ABB RobotStudio station: SCM_ExampleStation.rspag

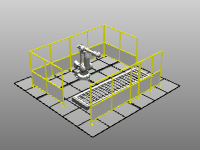
--- station ---
Station Station (saved by RobotStudio 6.4.7060.110)
Controller IRB4400_60_SCM_Example
  mechanical unit ROB_1: IRB4400_60_SCM_Example, 6 joints, base frame (0, 0, 0) mm
Layout (positions relative to the parent item):
  - Fence_2500 [graphiccomponentgroup, from Equipment\Fence_2500.rslib] at (-1042.5, 0, 0) mm
    - Body 1 [part, from Equipment\Fence_2500.rslib]
    - Body 2 [part, from Equipment\Fence_2500.rslib]
  - Fence_2500_2 [graphiccomponentgroup, from Equipment\Fence_2500.rslib] at (-1041.34, -2499.15, 0) mm
    - Body 1 [part, from Equipment\Fence_2500.rslib]
    - Body 2 [part, from Equipment\Fence_2500.rslib]
  - Fence_2500_3 [graphiccomponentgroup, from Equipment\Fence_2500.rslib] at (1452.87, 2467.85, 0) mm, rotated rx 0 ry 0 rz 89.7 deg
    - Body 1 [part, from Equipment\Fence_2500.rslib]
    - Body 2 [part, from Equipment\Fence_2500.rslib]
  - Fence_2500_4 [graphiccomponentgroup, from Equipment\Fence_2500.rslib] at (1428.43, -2470.87, 0) mm, rotated rx 0 ry 0 rz 90.52 deg
    - Body 1 [part, from Equipment\Fence_2500.rslib]
    - Body 2 [part, from Equipment\Fence_2500.rslib]
  - Conveyor 950 4000 h2 [part, from Equipment\Conveyor 950 4000 h2.rslib] at (2600.05, -2000, 0) mm, rotated rx 0 ry 0 rz 89.16 deg
  - Fence_2500_5 [graphiccomponentgroup, from Equipment\Fence_2500.rslib] at (3307.97, -2448.74, 0) mm
    - Body 1 [part, from Equipment\Fence_2500.rslib]
    - Body 2 [part, from Equipment\Fence_2500.rslib]
  - Fence_Gate [graphiccomponentgroup, from Equipment\Fence_Gate.rslib] at (3312.25, 0, 0) mm
    - Body 1 [part, from Equipment\Fence_Gate.rslib]
    - Body 2 [part, from Equipment\Fence_Gate.rslib]
    - Body 3 [part, from Equipment\Fence_Gate.rslib]
  - Fence_740 [graphiccomponentgroup, from Equipment\Fence_740.rslib] at (3289.25, 1511.78, 0) mm
    - Body 1 [part, from Equipment\Fence_740.rslib]
    - Body 2 [part, from Equipment\Fence_740.rslib]
  - IRB4400_60_SCM_Example [mechanism, from Robots\IRB4400_60_196_G_02.rslib] at (0, 0, 0) mm; joint values [0, 0, 0, 0, 0.5236, 0] (rad or m)

--- Backups/IRB4400_60_SCM_Example/RAPID/TASK1/PROGMOD/rollerData.mod ---
MODULE rollerData
  PERS num rollSizeIndex := 2;
  PERS num rollSize := 3.5;
  PERS num allowedRollSizes{5}:= [1.2,2.0, 3.5, 4.0, 6.6];
ENDMODULE

--- Backups/IRB4400_60_SCM_Example/RAPID/TASK1/PROGMOD/Routines.mod ---
MODULE Routines
	CONST jointtarget jntTgtHome:=[[0,0,0,0,0,0],[9E9,9E9,9E9,9E9,9E9,9E9]];
	CONST jointtarget jntTgtService:=[[0,0,0,0,0,0],[9E9,9E9,9E9,9E9,9E9,9E9]];

	PROC main()
		goHome;
	ENDPROC

	PROC goHome()
		MoveAbsJ jntTgtHome,v1000,fine,tool0\WObj:=wobj0;
	ENDPROC

	PROC goService()
		MoveAbsJ jntTgtHome,v1000,fine,tool0\WObj:=wobj0;
	ENDPROC

ENDMODULE

--- Backups/IRB4400_60_SCM_Example/RAPID/TASK1/SYSMOD/LINKEDM.sys ---
%%%
  VERSION:1
  LANGUAGE:ENGLISH
%%%

MODULE LINKEDM (SYSMODULE)

! FOLLOWER
!     Name of electronically linked follower axis used by operator at teach pendent.
      PERS string l_f_axis_name{5}       :=  ["",  "", "", "", ""];

!     Name of the mechanical unit for follower axis.
      PERS string l_f_mecunt_n{5}  :=  ["", "", "", "", ""];

!     Linked follower axis number in the mechanical unit (first axis in mech. unit is number 1).
      PERS num l_f_axis_no{5}      :=  [0,          0,   0,  0,  0];

! MASTER
!     Name of the mechanical unit for linked master axis.
      PERS string l_m_mecunt_n{5} :=  ["", "", "", "", ""];

!     Linked master axis number in the mechanical unit (first axis in mech. unit is number 1).
!     See axis number table in documentation for different master mechanical units.
      PERS num l_m_axis_no{5}     :=  [0,  0,  0,  0,  0];

! POSITION OFFSET
!     The increase of the allowed offset position between the master and follower
!     positions, used when starting AUTO mode. As soon as the offset is decreased
!     the old configurated parameter is used.
!     Example: 3 => the configurated value of allowed offset is increased 3 times.
      PERS num offset_ratio{5}       :=  [10,  10,   10,  10,  10];

! SPEED RATIO
!     Speed_ratio used in AUTO and JOG modes [ very_slow   slow    normal    fast]
!     Value 1 = max allowed manual speed.
      CONST num speed_ratio {20}      := [0.01, 0.01, 0.01, 0.01, 0.01,
                                          0.05, 0.05, 0.05, 0.05, 0.05,
                                          0.20, 0.20, 0.20, 0.20, 0.20,
                                          1.00, 1.00, 1.00, 1.00, 1.00];

! STEP SIZE
!     Displacement position used in JOG mode for each activation of positive or
!     negative movement.                  [very_short    short   normal   long]
!     Unit degees or meter.
      CONST num displacement {20}     := [0.001, 0.001, 0.001, 0.001, 0.001,
                                          0.005, 0.005, 0.005, 0.005, 0.005,
                                          0.020, 0.020, 0.020, 0.020, 0.020,
                                          0.100, 0.100, 0.100, 0.100, 0.100];


!-------------------------------------------------------------
 PROC Linked_m ()
      Linked_m_exe ;
 ENDPROC
ENDMODULE

--- Backups/IRB4400_60_SCM_Example/SYSPAR/EIO.cfg ---
EIO:CFG_1.0:6:1::
#
EIO_CROSS:

      -Name "AccessOK" -Res "diAccessOK" -Act1 "doGateRequestAccess"

      -Name "ConveyorForward" -Res "diConveyorForward" -Act1 "doConveyorForward"

      -Name "ConveyorReverse" -Res "diConveyorReverse" -Act1 "doConveyorReverse"

      -Name "LightCurtainStatus" -Res "diLightCurtainStatus"\
      -Act1 "doLightCurtainReset"
#
EIO_SIGNAL:

      -Name "doGateRequestAccess" -SignalType "DO" -Access "All"

      -Name "doConveyorForward" -SignalType "DO" -Access "All"

      -Name "doConveyorReverse" -SignalType "DO" -Access "All"

      -Name "doLightCurtainReset" -SignalType "DO" -Access "All"

      -Name "doMotorControl" -SignalType "DO" -Access "All"

      -Name "doConveyorSpeed" -SignalType "DO" -Access "All"

      -Name "diAccessOK" -SignalType "DI" -Access "All"

      -Name "diLightCurtainStatus" -SignalType "DI" -Access "All"

      -Name "diGateStatus" -SignalType "DI" -Access "All"

      -Name "diConveyorForward" -SignalType "DI" -Access "All"

      -Name "diConveyorReverse" -SignalType "DI" -Access "All"

      -Name "aoMotorSpeed" -SignalType "AO" -Access "All"
